// TwinCAT 3 PLC project pneumatic
// ProgramVersion: 3.1.4024.0
// libraries:
//   Tc2_Standard, * (Beckhoff Automation GmbH)
//   Tc2_System, * (Beckhoff Automation GmbH)
//   Tc3_Module, * (Beckhoff Automation GmbH)
// project tree:
//   GVLs/ GFY.TcGVL (not stored), GSS.TcGVL (not stored), GSYS.TcGVL (not stored)
//   / PlcTask.TcTTO
//   POUs/ Diff_n.TcPOU (not stored), FB_Backstep.TcPOU, Butter_ddq.TcPOU (not stored), Butter_dq.TcPOU (not stored), Butter_q.TcPOU, cmdTOxd.TcPOU (not stored), Diff.TcPOU (not stored), FBFY.TcPOU (not stored), FB_Backstep_ADRC.TcPOU (not stored), FB_BCRISENN.TcPOU (not stored), FB_DLADRC.TcPOU (not stored), FB_LADRC_BC.TcPOU (not stored), FB_SFVFPID.TcPOU, filter_oneMs.TcPOU (not stored), getAI.TcPOU (not stored), MAIN.TcPOU (not stored), PID.TcPOU, Sign.TcPOU (not stored), RISE.TcPOU (not stored), saturation.TcPOU (not stored), VFPID.TcPOU (not stored)
// real-time tasks:
//   TASK PlcTask: cycle T#1ms, priority 6, ADS port 350
// I/O:
//   DEVICE Device 1 (EtherCAT), AmsNetId 5.104.35.79.2.1
//     Term 1 (EK1200) [EK1200-5000 EtherCAT Power supply (2A E-Bus)]
//       Term 2 (EL1889) [EL1889 16Ch. Dig. Input 24V, 3ms, negative]
//       Term 3 (EL2809) [EL2809 16Ch. Dig. Output 24V, 0.5A]
//       Term 4 (EL3174) [EL3174 4Ch. Ana. Input +/-10V Diff., +/-20mA SingleEnded, 16 Bit]
//       Term 5 (EL3174) [EL3174 4Ch. Ana. Input +/-10V Diff., +/-20mA SingleEnded, 16 Bit]
//       Term 6 (EL4104) [EL4104 4Ch. Ana. Output 0-10V, 16bit]
//       Term 7 (EL4104) [EL4104 4Ch. Ana. Output 0-10V, 16bit]
//       Term 8 (EL4124) [EL4124 4Ch. Ana. Output 4-20mA, 16bit]
//       Term 9 (EL9011) [EL9011 End Terminal]
//   DEVICE Device 3 (NOV-DP-RAM)
// variable links:
//   pneumatic/pneumatic Instance <-> Device 1 (EtherCAT)/Term 1 (EK1200)/Term 2 (EL1889)
//     PlcTask Inputs/MAIN.shenchu <-> Channel 1/Input
//     PlcTask Inputs/MAIN.suohui <-> Channel 2/Input
//   pneumatic/pneumatic Instance <-> Device 1 (EtherCAT)/Term 1 (EK1200)/Term 3 (EL2809)
//     PlcTask Outputs/MAIN.JZF <-> Channel 2/Output
//   pneumatic/pneumatic Instance <-> Device 1 (EtherCAT)/Term 1 (EK1200)/Term 4 (EL3174)
//     PlcTask Inputs/MAIN.FY.BMQ <-> AI Standard Channel 3/Value
//     PlcTask Inputs/MAIN.FY.WY <-> AI Standard Channel 4/Value
//     PlcTask Inputs/MAIN.FY.YL1 <-> AI Standard Channel 1/Value
//     PlcTask Inputs/MAIN.FY.YL2 <-> AI Standard Channel 2/Value
//   pneumatic/pneumatic Instance <-> Device 1 (EtherCAT)/Term 1 (EK1200)/Term 6 (EL4104)
//     PlcTask Outputs/MAIN.FY.BLFKZ <-> AO Output Channel 2/Analog output

CONFIGURATION pneumatic
    RESOURCE PLC ON TwinCAT3
        TASK PlcTask(INTERVAL := T#1ms, PRIORITY := 6);
        PROGRAM MAIN WITH PlcTask : MAIN;
    END_RESOURCE
END_CONFIGURATION

// ---- POUs/FB_Backstep.TcPOU
FUNCTION_BLOCK FB_Backstep
VAR_INPUT
	x1d:REAL;
	x1:REAL;  
	x2:REAL;  
	x3:REAL;  
	Amp:REAL;
	krise:REAL;
	BC_up:REAL;
	BC_down:REAL;
	cyct:REAL;
	k1:REAL;
	f1:REAL;
	f2:REAL;
	k2:REAL;
	k3:REAL;
	L_d:REAL;
	b0:REAL;
	w2:REAL;
	w3:REAL;
	kr1:REAL;
	kr2:REAL;
	beta1:REAL;
	beta2:REAL;
	M:REAL;  
	aw:REAL; 
	daw:REAL; 
	d1:REAL; 
	u_L:REAL; 
END_VAR
VAR_OUTPUT
	z1:REAL;
	a1:REAL;
	ar1:REAL;
	z2:REAL;
	dz2:REAL;
	a2:REAL;
	ar2:REAL;
	z3:REAL;
	u:REAL;
	u_BC:REAL;
	da1:REAL;
	dda1:REAL;
	da2:REAL;
	da2_BC:REAL;
	ed1:REAL;
	ed2:REAL;
END_VAR
VAR
	Feed:REAL:=0;
	L_x1d:REAL:=0;
	LL_x1d:REAL:=0;
	dz1:REAL;
	dx1d:REAL;
	L_dx1d:REAL:=0;
	ddx1d:REAL:=0;
	L_ddx1d:REAL:=0;
	dddx1d:REAL:=0;
	
	sign1:REAL:=0;
	Inte11:REAL:=0;
	Inte12:REAL:=0;
	Inte21:REAL:=0;
	Inte22:REAL:=0;
	
	Tf1:REAL;
	x2f:REAL;
	L_x2f:REAL:=0;
	L_a2:REAL:=0;
	x3f:REAL;
	L_x3f:REAL:=0;
	
	Tf2:REAL;
	
	edx1:REAL;
	ex1:REAL:=0;
	ex2:REAL:=0;
	edx2:REAL;
	edd1:REAL;
	
	ex3:REAL:=0;
	edx3:REAL;
	edd2:REAL;
	
	kr1c:REAL;
	kr2c:REAL;
	beta1c:REAL;
	beta2c:REAL;
END_VAR


edx1:=ex2-3*w2*(ex1-x1);
edx2:=(x3-aw)/M*L_d+ed1-3*w2*w2*(ex1-x1);
edd1:=-w2*w2*w2*(ex1-x1);

edx3:=b0*u_L+ed2-2*w3*(ex3-x3);
edd2:=-w3*w3*(ex3-x3);

ex1:=ex1+edx1*cyct;
ex2:=ex2+edx2*cyct;
ex3:=ex3+edx3*cyct;
ed2:=ed2+edd2*cyct;
ed1:=ed1+edd1*cyct;

z1:=x1-x1d;
dx1d:=(x1d-L_x1d)/cyct;
dz1:=ex2-dx1d;
L_x1d:=x1d;
a1:=dx1d-k1*z1;

z2:=ex2-a1;
ddx1d:=(dx1d-L_dx1d)/cyct;
L_dx1d:=dx1d;
dddx1d:=0*(ddx1d-L_ddx1d)/cyct;
L_ddx1d:=ddx1d;

da1:=ddx1d-k1*(ex2-dx1d);

//变rise1
kr1c:=kr1*EXPT(2.71828,-(Amp-ABS(krise)));
beta1c:=beta1*EXPT(2.71828,-(Amp-ABS(krise)));

ar1:=-M*kr1c*z2-(kr1c*k2*Inte11+beta1c*Inte12);

IF GFY.BC_kr1=0 THEN
	Inte11:=0;
	Inte12:=0;
ELSE
	Inte11:=Inte11+z2*cyct;
	Inte12:=Inte12+Sign(x:=z2)*cyct;
END_IF

a2:=(-k2*z2+M*da1-M*ed1+ar1)/L_d+aw;
//a2:=aw+M*da1-k2*z2+ar1;

dda1:=dddx1d-k1*(edx2-ddx1d);
dz2:=edx2-da1;

z3:=x3-a2;


da2_BC:=(-k2*dz2+M*dda1-M*edd1)/L_d+daw;;


kr2c:=kr2*EXPT(2.71828,-(Amp-ABS(krise)));
beta2c:=beta2*EXPT(2.71828,-(Amp-ABS(krise)));

ar2:=-kr2c*z3-(kr2c*k3*Inte21+beta2c*Inte22);

IF GFY.BC_kr2=0 THEN
	Inte21:=0;
	Inte22:=0;
ELSE
	Inte21:=Inte21+z3*cyct;
	Inte22:=Inte22+Sign(x:=z3)*cyct;
END_IF

u_BC:=(-k3*z3+da2_BC-ed2+ar2)/b0;
u_BC:=saturation(upLMT:=BC_up,downLMT:=BC_down,input:=u_BC);

END_FUNCTION_BLOCK

// ---- POUs/Butter_q.TcPOU
FUNCTION_BLOCK Butter_q  //位移/角度的二阶巴特沃斯滤波器
VAR_INPUT
	But_u:REAL;
	But_wn:REAL;
	But_Ts:REAL;
END_VAR
VAR_OUTPUT
	But_y:REAL;
END_VAR
VAR
	aa:REAL:=0;
	last_y:REAL:=0;
	llast_y:REAL:=0;
END_VAR

But_y:=(But_u*But_wn*But_wn*But_Ts*But_Ts)/(1+But_wn*But_wn*But_Ts*But_Ts+SQRT(2)*But_wn*But_Ts)
      +last_y*(2+SQRT(2)*But_wn*But_Ts)/(1+But_wn*But_wn*But_Ts*But_Ts+SQRT(2)*But_wn*But_Ts)
	  -llast_y/(1+But_wn*But_wn*But_Ts*But_Ts+SQRT(2)*But_wn*But_Ts);

aa:=last_y;  
last_y:=But_y; 
llast_y:=aa;

END_FUNCTION_BLOCK

// ---- POUs/FB_SFVFPID.TcPOU
FUNCTION_BLOCK FB_SFVFPID

VAR_INPUT  
    RespectValue: REAL;//期望值
	RealValue   : REAL;//实际值
	
	PID_Kv:REAL;
	PID_Kp:REAL;
	PID_Ki:REAL;
	PID_Kd:REAL;
	KF:REAL;
	F:REAL;
	KdF:REAL;
	dF:REAL;
	Kdx:REAL;
	dx:REAL;
	upLMT_int:REAL;     //抗积分饱和
	downLMT_int:REAL;   //抗积分饱和
	upLMT_out:REAL;     //输出限幅
	downLMT_out:REAL;   //输出限幅

	PID_Integral     : REAL := 0.0;//定义积分项
END_VAR
VAR_OUTPUT
	P_PART:REAL;
	I_PART:REAL;
	D_PART:REAL;
	V_PART:REAL;
	SFVFPID_Out:REAL;
	
END_VAR
VAR
	PID_Error        : REAL := 0.0;//偏差
    PID_LastError    : REAL := 0.0;//上次偏差
	PID_L_LastError  : REAL := 0.0;//上上次偏差
	PID_Proportion   : REAL := 0.0;//定义比例项
	PID_VF           : REAL:= 0.0;  //定义速度前馈项
	PID_Differential : REAL;       //定义微分项
	PID_L_SetValue   : REAL := 0.0;//上次指令
	PID_Temp         : REAL;       //输出
END_VAR

PID_Error:=RespectValue-RealValue;          //偏差=期望值-实际值
PID_Proportion:=PID_Error;                         //比例项=偏差
PID_Integral := PID_Integral+PID_Ki*PID_Error;			//积分项=偏差累积

//抗积分饱和
PID_Integral:=saturation(upLMT:=upLMT_int , downLMT:=downLMT_int , input:=PID_Integral );
PID_VF:=RespectValue-PID_L_SetValue;               //速度前馈项=指令-上次指令
PID_Differential:=PID_Error-PID_LastError;         //微分项=偏差-上次偏差

P_PART:=PID_Kp*PID_Proportion;
I_PART:=PID_Integral;
D_PART:=PID_Kd*PID_Differential;
V_PART:=PID_Kv*PID_VF;
PID_Temp:=PID_Kp*PID_Proportion+PID_Integral+PID_Kd*PID_Differential+PID_Kv*PID_VF; //PID控制

PID_L_SetValue:=RespectValue;
PID_LastError:=PID_Error;
//输出限幅
PID_Temp:=PID_Temp-KF*F-KdF*dF-Kdx*dx;
SFVFPID_Out:=saturation(upLMT:=upLMT_out , downLMT:=downLMT_out , input:=PID_Temp );

END_FUNCTION_BLOCK

// ---- POUs/PID.TcPOU
FUNCTION_BLOCK PID
VAR_INPUT
	RespectValue: REAL;//期望值
	RealValue   : REAL;//实际值
	
	PID_Kp:REAL;
	PID_Ki:REAL;
	PID_Kd:REAL;
	upLMT_int:REAL;     //抗积分饱和
	downLMT_int:REAL;   //抗积分饱和
	upLMT_out:REAL;     //输出限幅
	downLMT_out:REAL;   //输出限幅
	
	temp:REAL;
	PID_Integral     : REAL := 0.0;//定义积分项
END_VAR
VAR_OUTPUT
	P_PART:REAL;
	I_PART:REAL;
	D_PART:REAL;
	PID_Out:REAL;
	
END_VAR
VAR
	PID_Error        : REAL := 0.0;//偏差
    PID_LastError    : REAL := 0.0;//上次偏差
	PID_L_LastError  : REAL := 0.0;//上上次偏差
	PID_Proportion   : REAL := 0.0;//定义比例项
	
	PID_Differential : REAL;       //定义微分项
	PID_L_SetValue   : REAL := 0.0;//上次指令
	PID_Temp         : REAL;       //输出
END_VAR

PID_Error:=RespectValue-RealValue;          //偏差=期望值-实际值
PID_Proportion:=PID_Error;                         //比例项=偏差
PID_Integral := PID_Integral+PID_Ki*PID_Error;			//积分项=偏差累积

//抗积分饱和
PID_Integral:=saturation(upLMT:=upLMT_int , downLMT:=downLMT_int , input:=PID_Integral );

PID_Differential:=PID_Error-PID_LastError;         //微分项=偏差-上次偏差

P_PART:=PID_Kp*PID_Proportion;
I_PART:=PID_Integral;
D_PART:=PID_Kd*PID_Differential;
PID_Temp:=PID_Kp*PID_Proportion+PID_Integral+PID_Kd*PID_Differential; //PID控制

PID_L_SetValue:=RespectValue;
PID_LastError:=PID_Error;
//输出限幅
PID_Out:=saturation(upLMT:=upLMT_out , downLMT:=downLMT_out , input:=PID_Temp );

END_FUNCTION_BLOCK
